// TwinCAT 3 PLC project Untitled1
// ProgramVersion: 3.1.4023.0
// libraries:
//   Tc2_Standard, * (Beckhoff Automation GmbH)
//   Tc2_System, * (Beckhoff Automation GmbH)
//   Tc3_Module, * (Beckhoff Automation GmbH)
// project tree:
//   / PlcTask.TcTTO
//   POUs/ MAIN.TcPOU
// real-time tasks:
//   TASK PlcTask: cycle T#1ms, priority 20, ADS port 350

CONFIGURATION Untitled1
    RESOURCE PLC ON TwinCAT3
        TASK PlcTask(INTERVAL := T#1ms, PRIORITY := 20);
        PROGRAM MAIN WITH PlcTask : MAIN;
    END_RESOURCE
END_CONFIGURATION

// ---- POUs/MAIN.TcPOU
PROGRAM MAIN
VAR
	ton_a 	: TON := (PT:=T#1S);
	ton_b	: TON := (PT:=T#0.1S);
	n_cnt_a : UINT := 1;  // 1/s
	n_cnt_b : UINT := 2; // 1/100ms
	n_cnt_c : UINT := 3; // 1/ms
END_VAR

ton_a(IN:= NOT ton_a.Q);
ton_b(IN:= NOT ton_b.Q);

IF ton_a.Q THEN
	n_cnt_a := n_cnt_a + 1;
END_IF

IF ton_b.Q THEN
	n_cnt_b := n_cnt_b + 1;
END_IF

n_cnt_c := n_cnt_c + 1;

END_PROGRAM
